TYPE stStationInfo :
STRUCT
	StationProcessTime : TIME;
	StationPosition : MC_LREAL;
	StationStatus : stStationStatus;
END_STRUCT
END_TYPE

(* stored: Version 1.1.0.1
   DUT stStationInfo: Id {7dd8a7ee-b816-4ef5-ad77-227cfdfcc86f} *)
